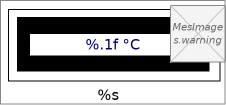
VISUALIZATION VISU_TEMPRO_PLUS_90  // 226x105
VAR_IN_OUT
	m_Input_RECHAUF : BLOCK_TEMPRO90_ANA;
END_VAR
    Rectangle (17,17 192x54), colour toggle: m_Input_RECHAUF.STATE_PowerOn
    Rectangle (8,9 212x72), invisible if: NOT (m_Input_RECHAUF.AUTOR_PowerOn_IHM OR m_Input_RECHAUF.AUTOR_PowerOff_IHM) OR NOT PRG_User.ACTU_USER.MAINTENANCE
        tap m_Input_RECHAUF.M_PowerOn
    Rectangle (88,85 41x20), "%s", text variable: m_Input_RECHAUF.MNEMO
    RoundedRectangle (29,33 168x23), "%.1f °C", text variable: m_Input_RECHAUF.STATE_Temp
    Image (170,5 56x57), invisible if: NOT m_Input_RECHAUF.STATE_Nok, image: MesImages.warning
END_VISUALIZATION

// ---- Visualizations/Symbole/STACKER/VISU_SUBSTRAT_NO_NUM.TcVIS
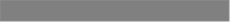
VISUALIZATION VISU_SUBSTRAT_NO_NUM  // 230x22
VAR_IN_OUT
	m_Input_MAP: STRUCT_MACHINE;
END_VAR
VAR_INPUT
	m_Input_NUM_CHAMBER : UDINT;
	m_Input_NUM_STATION : UDINT;
END_VAR
    Rectangle (0,0 228x20), invisible if: NOT m_Input_MAP.CHAMBER[m_Input_NUM_CHAMBER].STATION[m_Input_NUM_STATION].STATE_Unloaded
    Rectangle (0,0 228x20), invisible if: NOT m_Input_MAP.CHAMBER[m_Input_NUM_CHAMBER].STATION[m_Input_NUM_STATION].STATE_Loaded
    Rectangle (0,0 228x20), invisible if: m_Input_MAP.CHAMBER[m_Input_NUM_CHAMBER].STATION[m_Input_NUM_STATION].STATE_Loaded OR m_Input_MAP.CHAMBER[m_Input_NUM_CHAMBER].STATION[m_Input_NUM_STATION].STATE_Unloaded
END_VISUALIZATION

// ---- Visualizations/Symbole/VANNES/VISU_VANNE_2P_H.TcVIS
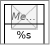
VISUALIZATION VISU_VANNE_2P_H  // 50x45
VAR_IN_OUT
	m_Input_VANNE : BLOCK_ACTUATOR;
END_VAR
    Rectangle (4,4 40x40), invisible if: TRUE
    Polygon (0,0)
    Rectangle (-1,25 50x20), "%s", text variable: m_Input_VANNE.MNEMO
    Polygon (0,0), colour toggle: (m_Input_VANNE.STATE_ON) <> 0, invisible if: NOT (m_Input_VANNE.STATE_OFF OR m_Input_VANNE.STATE_ON)
    Image (11,4 26x25), invisible if: NOT m_Input_VANNE.STATE_Nok, image: MesImages.warning
    Rectangle (4,4 40x20), invisible if: NOT (m_Input_VANNE.Autor_ON_IHM OR m_Input_VANNE.Autor_OFF_IHM) OR NOT PRG_User.ACTU_USER.MAINTENANCE
        tap m_Input_VANNE.M_ON
END_VISUALIZATION

// ---- Visualizations/Symbole/VANNES/VISU_VANNE_2P_H_ACT2.TcVIS
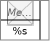
VISUALIZATION VISU_VANNE_2P_H_ACT2  // 50x41
VAR_IN_OUT
	m_Input_VANNE : BLOCK_ACTUATOR2;
END_VAR
    Rectangle (0,0 40x40), invisible if: TRUE
    Polygon (0,0)
    Rectangle (-5,21 50x20), "%s", text variable: m_Input_VANNE.MNEMO
    Polygon (0,0), colour toggle: (m_Input_VANNE.STATE_ON) <> 0, invisible if: NOT (m_Input_VANNE.STATE_OFF OR m_Input_VANNE.STATE_ON)
    Image (7,0 26x25), invisible if: NOT m_Input_VANNE.STATE_Nok, image: MesImages.warning
    Rectangle (0,0 40x20), invisible if: NOT (m_Input_VANNE.Autor_ON_IHM OR m_Input_VANNE.Autor_OFF_IHM) OR NOT PRG_User.ACTU_USER.MAINTENANCE
        tap m_Input_VANNE.M_ON
END_VISUALIZATION

// ---- Visualizations/Symbole/VANNES/VISU_VANNE_2P_V.TcVIS
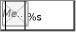
VISUALIZATION VISU_VANNE_2P_V  // 76x32
VAR_IN_OUT
	m_Input_VANNE : BLOCK_ACTUATOR;
END_VAR
    Rectangle (0,0 74x30), invisible if: TRUE
    Polygon (50,0)
    Polygon (50,0), colour toggle: (m_Input_VANNE.STATE_ON), invisible if: NOT (m_Input_VANNE.STATE_OFF OR m_Input_VANNE.STATE_ON) AND NOT PRG_USER.ACTU_USER.MAINTENANCE
    Rectangle (24,7 50x20), "%s", text variable: m_Input_VANNE.MNEMO
    Image (2,1 26x25), invisible if: NOT m_Input_VANNE.STATE_Nok, image: MesImages.warning
    Rectangle (5,0 20x30), invisible if: NOT (m_Input_VANNE.Autor_ON_IHM OR m_Input_VANNE.Autor_OFF_IHM) OR NOT PRG_User.ACTU_USER.MAINTENANCE
        tap m_Input_VANNE.M_ON
END_VISUALIZATION

// ---- Visualizations/Symbole/VANNES/VISU_VANNE_2P_V_ACT2.TcVIS
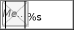
VISUALIZATION VISU_VANNE_2P_V_ACT2  // 74x30
VAR_IN_OUT
	m_Input_VANNE : BLOCK_ACTUATOR2;
END_VAR
    Rectangle (0,0 74x30), invisible if: TRUE
    Polygon (50,0)
    Polygon (50,0), colour toggle: (m_Input_VANNE.STATE_ON), invisible if: NOT (m_Input_VANNE.STATE_OFF OR m_Input_VANNE.STATE_ON) AND NOT PRG_USER.ACTU_USER.MAINTENANCE
    Rectangle (24,7 50x20), "%s", text variable: m_Input_VANNE.MNEMO
    Image (2,1 26x25), invisible if: NOT m_Input_VANNE.STATE_Nok, image: MesImages.warning
    Rectangle (5,0 20x30), invisible if: NOT (m_Input_VANNE.Autor_ON_IHM OR m_Input_VANNE.Autor_OFF_IHM) OR NOT PRG_User.ACTU_USER.MAINTENANCE
        tap m_Input_VANNE.M_ON
END_VISUALIZATION

// ---- Visualizations/Symbole/VANNES/VISU_VANNE_2P_V_NoPilot.TcVIS
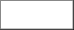
VISUALIZATION VISU_VANNE_2P_V_NoPilot  // 74x30
    Rectangle (0,0 74x30), invisible if: TRUE
    Polygon (50,0)
END_VISUALIZATION

// ---- Visualizations/Symbole/VANNES/VISU_VANNE_3P_H.TcVIS
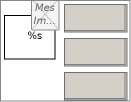
VISUALIZATION VISU_VANNE_3P_H  // 131x102
VAR_IN_OUT
	m_Input_Vanne	:	BLOCK_VVAT_3P;
END_VAR
    Rectangle (4,15 51x44), invisible if: TRUE
    Polygon (0,0), colour toggle: m_Input_Vanne.STATE_Lam
    Rectangle (13,25 44x21), "%s", text variable: m_Input_Vanne.MNEMO
    Polygon (0,0), colour toggle: m_Input_Vanne.STATE_On, invisible if: NOT (m_Input_Vanne.STATE_Off or m_Input_Vanne.STATE_On)
    Button (64,4 63x28), input disabled if: NOT m_Input_Vanne.AUTOR_On_IHM OR NOT .PRG_USER.ACTU_USER.MAINTENANCE, text list: 'TextList_VVAT_3P', text index: 0
        OnMouseClick: toggle m_Input_Vanne.M_On
    Button (64,38 63x28), input disabled if: NOT m_Input_Vanne.AUTOR_Lam_IHM OR NOT .PRG_USER.ACTU_USER.MAINTENANCE, text list: 'TextList_VVAT_3P', text index: 2
        OnMouseClick: toggle m_Input_Vanne.M_Lam
    Button (64,72 63x28), input disabled if: NOT m_Input_Vanne.AUTOR_Off_IHM OR NOT .PRG_USER.ACTU_USER.MAINTENANCE, text list: 'TextList_VVAT_3P', text index: 1
        OnMouseClick: toggle m_Input_Vanne.M_Off
    Image (31,-2 28x32), invisible if: NOT m_Input_Vanne.STATE_Nok, image: MesImages.warning
END_VISUALIZATION

// ---- Visualizations/Symbole/VANNES/VISU_VANNE_ASS_H.TcVIS
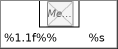
VISUALIZATION VISU_VANNE_ASS_H  // 118x49
VAR_IN_OUT
	m_Input_VANNE : BLOCK_VVAT_650_NO;
END_VAR

VAR_INPUT
	m_Input_NumFrame_Manu:	USINT;		(*numéro de frame à afficher dans le synoptique MANUEL*)
END_VAR
    Rectangle (0,0 118x49), invisible if: TRUE
    Polygon (0,0), colour toggle: m_Input_VANNE.STATE_Lam
    Rectangle (76,28 41x20), "%s", text variable: m_Input_VANNE.MNEMO
    Polygon (0,0), colour toggle: m_Input_VANNE.STATE_On, invisible if: NOT (m_Input_VANNE.STATE_Off OR m_Input_VANNE.STATE_On)
    Ellipse (54,2 10x10), colour toggle: m_Input_VANNE.STATE_Ok, invisible if: NOT m_Input_VANNE.STATE_Ok
    Rectangle (1,28 77x20), "%1.1f%%", text variable: m_Input_VANNE.STATE_Position
    Image (47,1 26x25), invisible if: NOT m_Input_VANNE.STATE_Nok, image: MesImages.warning
    Rectangle (39,0 40x27), invisible if: NOT m_Input_VANNE.MANUAL
        OnMouseClick: execute { .VISU_INDEX_MANU := m_Input_NumFrame_Manu; }
        OnMouseClick: change screen: SYN_MANUEL
END_VISUALIZATION

// ---- Visualizations/Symbole/VANNES/VISU_VANNE_ASS_H_MANU.TcVIS
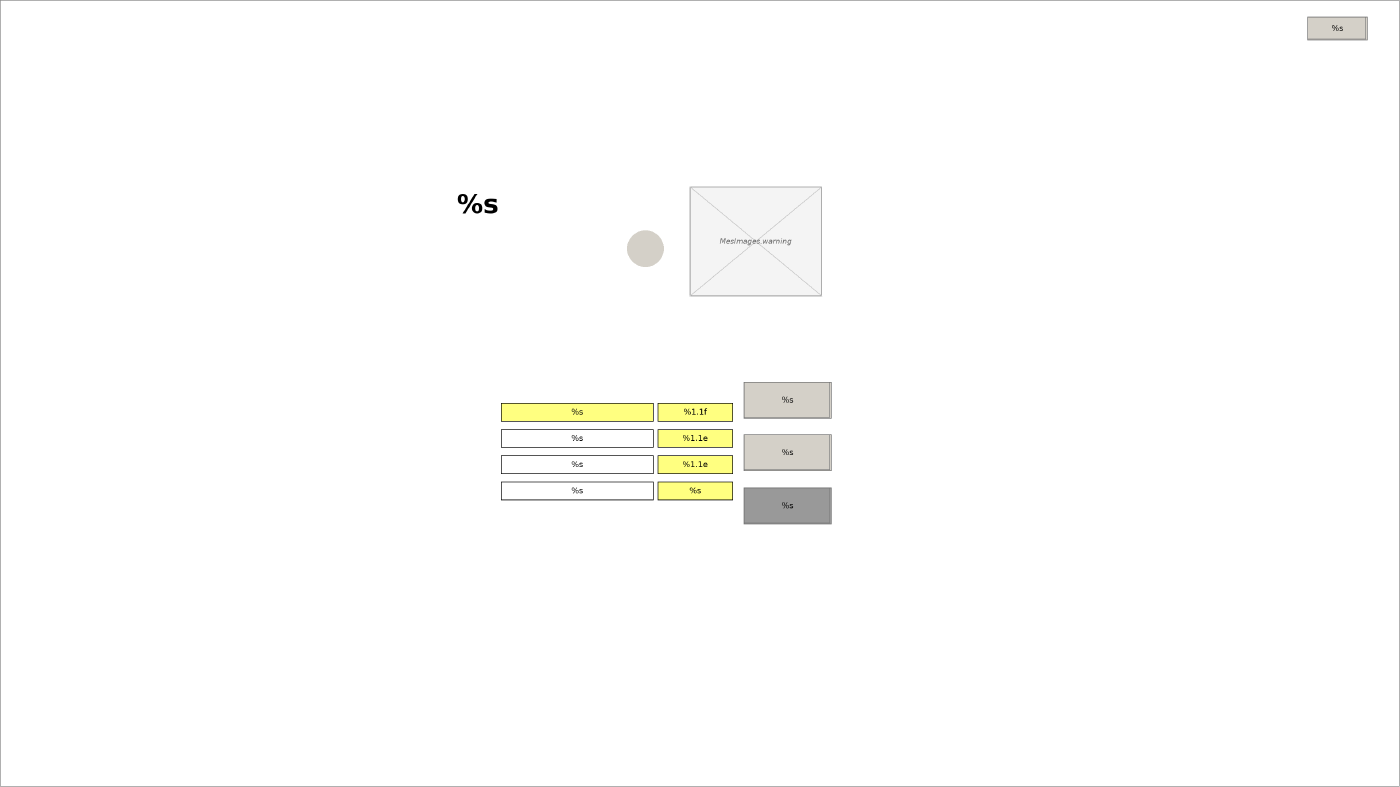
VISUALIZATION VISU_VANNE_ASS_H_MANU  // 1920x1080
VAR_IN_OUT
	m_Input_Vanne:		BLOCK_VVAT_650_NO;
	m_Input_State_Manu:	BOOL;
END_VAR
    Button (1793,23 82x32), "%s", text list: 'TextList_Basiques', text index: 8
        OnMouseClick: change screen: Previous 
        OnMouseClick: execute { .VISU_INDEX_MANU := 0; }
    Polygon (0,0), colour toggle: m_Input_VANNE.STATE_Lam
    Rectangle (573,246 165x68), "%s", text variable: m_Input_VANNE.MNEMO
    Polygon (0,0), colour toggle: m_Input_VANNE.STATE_On, invisible if: NOT (m_Input_VANNE.STATE_Off OR m_Input_VANNE.STATE_On)
    Ellipse (860,316 50x50), colour toggle: m_Input_VANNE.STATE_Ok
    Image (946,256 181x150), invisible if: NOT m_Input_VANNE.STATE_Nok, image: MesImages.warning
    Button (1020,524 120x50), "%s", input disabled if: NOT m_Input_Vanne.AUTOR_On_IHM OR NOT .PRG_USER.ACTU_USER.MAINTENANCE, text list: 'TextList_VVAT_3P', text index: 0
        toggle m_Input_Vanne.M_On
    Button (1020,596 120x50), "%s", input disabled if: NOT m_Input_Vanne.AUTOR_Off_IHM OR NOT .PRG_USER.ACTU_USER.MAINTENANCE, text list: 'TextList_VVAT_3P', text index: 1
        toggle m_Input_Vanne.M_Off
    Button (1020,669 120x50), "%s", input disabled if: NOT m_Input_Vanne.AUTOR_Lam_IHM OR NOT .PRG_USER.ACTU_USER.MAINTENANCE, text list: 'TextList_VVAT_3P', text index: 2
        toggle m_Input_Vanne.M_Lam
    RoundedRectangle (687,553 209x25), "%s", invisible if: NOT m_Input_Vanne.PRM_Mode, input disabled if: NOT .PRG_USER.ACTU_USER.MAINTENANCE OR NOT m_Input_State_Manu OR NOT m_Input_Vanne.PRM_Mode, text list: 'TextList_VVAT_650_ETHERCAT', text index: 8
        OnMouseClick: toggle m_Input_Vanne.PRM_Mode
    RoundedRectangle (687,553 209x25), "%s", invisible if: m_Input_Vanne.PRM_Mode, input disabled if: NOT .PRG_USER.ACTU_USER.MAINTENANCE OR NOT m_Input_State_Manu OR m_Input_Vanne.PRM_Mode, text list: 'TextList_VVAT_650_ETHERCAT', text index: 7
        OnMouseClick: toggle m_Input_Vanne.PRM_Mode
    RoundedRectangle (687,589 209x25), "%s", invisible if: NOT m_Input_Vanne.PRM_Mode, text list: 'TextList_VVAT_650_ETHERCAT', text index: 4
    RoundedRectangle (687,625 209x25), "%s", invisible if: NOT m_Input_Vanne.PRM_Mode, text list: 'TextList_VVAT_650_ETHERCAT', text index: 5
    RoundedRectangle (687,661 209x25), "%s", invisible if: NOT m_Input_Vanne.PRM_Mode, text list: 'TextList_VVAT_650_ETHERCAT', text index: 6
    RoundedRectangle (902,661 103x25), "%s", text variable: m_Input_Vanne.PRM_Tim_W_Pr, invisible if: NOT m_Input_Vanne.PRM_Mode, input disabled if: NOT m_Input_Vanne.PRM_Mode
        OnMouseClick: write the text variable via Edit
    RoundedRectangle (902,625 103x25), "%1.1e", text variable: m_Input_Vanne.PRM_W_Pr_HI, invisible if: NOT m_Input_Vanne.PRM_Mode, input disabled if: NOT m_Input_Vanne.PRM_Mode
        OnMouseClick: write the text variable via InputWithLimits, min 0, max 1000
    RoundedRectangle (902,589 103x25), "%1.1e", text variable: m_Input_Vanne.PRM_W_Pr_LO, invisible if: NOT m_Input_Vanne.PRM_Mode, input disabled if: NOT m_Input_Vanne.PRM_Mode
        OnMouseClick: write the text variable via InputWithLimits, min 0, max 1000
    RoundedRectangle (902,553 103x25), "%1.1e", text variable: m_Input_Vanne.PRM_Pression, invisible if: NOT m_Input_Vanne.PRM_Mode, input disabled if: NOT m_Input_Vanne.PRM_Mode
        OnMouseClick: write the text variable via InputWithLimits, min 0, max 1000
    RoundedRectangle (902,553 103x25), "%1.1f", text variable: m_Input_Vanne.PRM_Position, invisible if: m_Input_Vanne.PRM_Mode, input disabled if: m_Input_Vanne.PRM_Mode
        OnMouseClick: write the text variable via InputWithLimits, min 0, max 100
END_VISUALIZATION

// ---- Visualizations/Symbole/VANNES/VISU_VANNE_ASS_VAT653_ETHERCAT.TcVIS
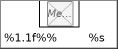
VISUALIZATION VISU_VANNE_ASS_VAT653_ETHERCAT  // 118x49
VAR_IN_OUT
	m_Input_VANNE : BLOCK_VVAT_653_ETHERCAT;
END_VAR

VAR_INPUT
	m_Input_NumFrame_Manu:	USINT;		(*numéro de frame à afficher dans le synoptique MANUEL*)
END_VAR
    Rectangle (0,0 118x49), invisible if: TRUE
    Polygon (0,0), colour toggle: m_Input_VANNE.STATE_Lam
    Rectangle (76,28 41x20), "%s", text variable: m_Input_VANNE.MNEMO
    Polygon (0,0), colour toggle: m_Input_VANNE.STATE_On, invisible if: NOT (m_Input_VANNE.STATE_Off OR m_Input_VANNE.STATE_On)
    Ellipse (54,2 10x10), colour toggle: m_Input_VANNE.STATE_Ok, invisible if: NOT m_Input_VANNE.STATE_Ok
    Rectangle (1,28 77x20), "%1.1f%%", text variable: m_Input_VANNE.STATE_Position
    Image (47,1 26x25), invisible if: NOT m_Input_VANNE.STATE_Nok, image: MesImages.warning
    Rectangle (39,0 40x27), invisible if: NOT m_Input_VANNE.MANUAL
        OnMouseClick: execute { .VISU_INDEX_MANU := m_Input_NumFrame_Manu; }
        OnMouseClick: change screen: SYN_MANUEL
END_VISUALIZATION

// ---- Visualizations/Symbole/VANNES/VISU_VANNE_ASS_VAT653_ETHERCAT_MANU.TcVIS
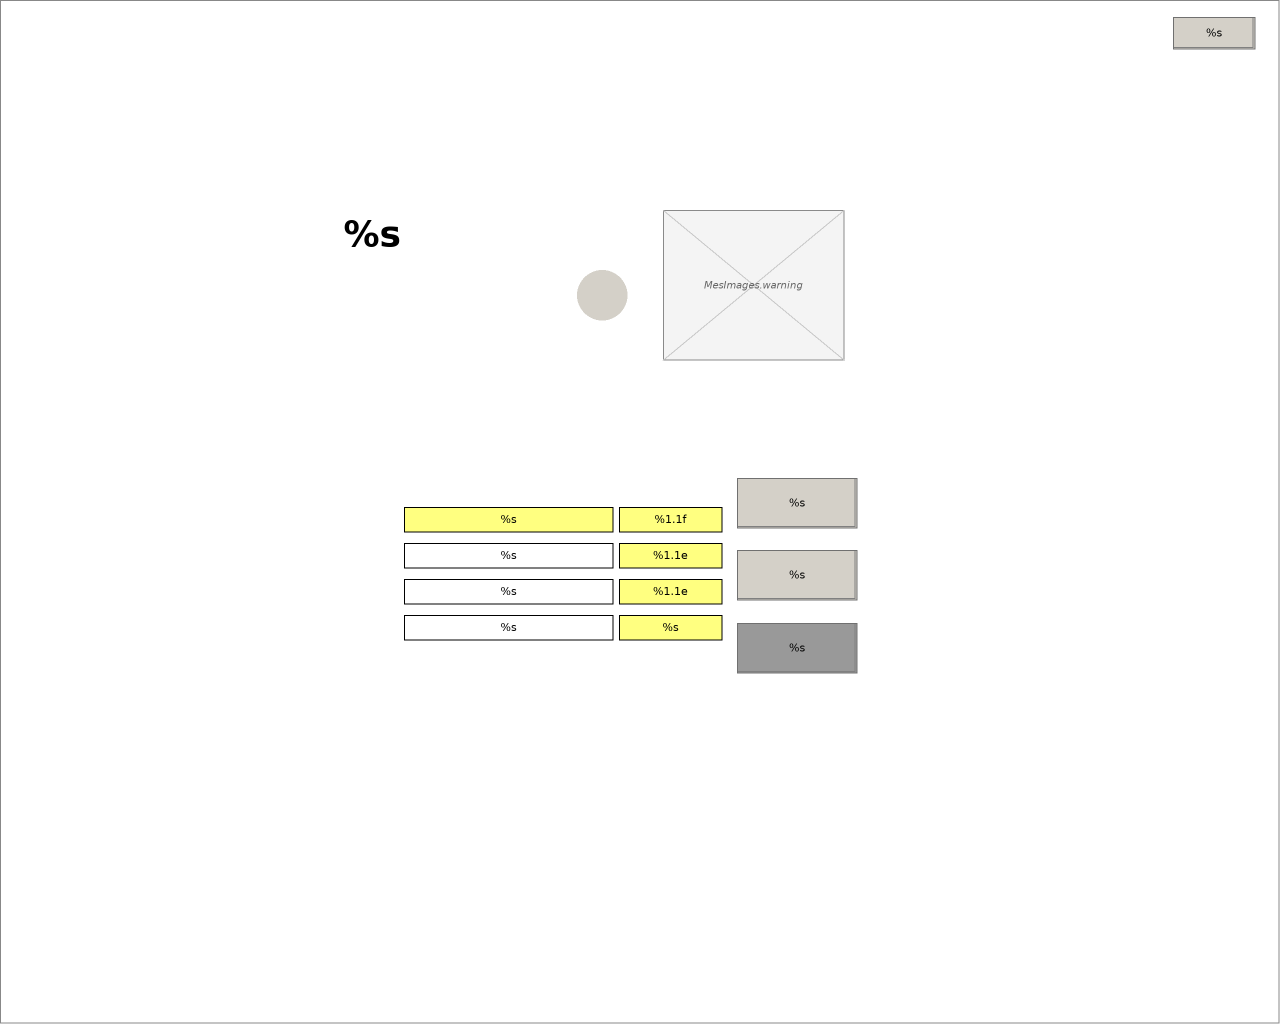
VISUALIZATION VISU_VANNE_ASS_VAT653_ETHERCAT_MANU  // 1280x1024
VAR_IN_OUT
	m_Input_Vanne:		BLOCK_VVAT_653_ETHERCAT;
	m_Input_State_Manu:	BOOL;
END_VAR
    Button (1173,17 82x32), "%s", text list: 'TextList_Basiques', text index: 8
        OnMouseClick: change screen: Previous 
        OnMouseClick: execute { .VISU_INDEX_MANU := 0; }
    Polygon (0,0), colour toggle: m_Input_VANNE.STATE_Lam
    Rectangle (290,200 165x68), "%s", text variable: m_Input_VANNE.MNEMO
    Polygon (0,0), colour toggle: m_Input_VANNE.STATE_On, invisible if: NOT (m_Input_VANNE.STATE_Off OR m_Input_VANNE.STATE_On)
    Ellipse (577,270 50x50), colour toggle: m_Input_VANNE.STATE_Ok, invisible if: NOT m_Input_VANNE.STATE_Ok
    Image (663,210 181x150), invisible if: NOT m_Input_VANNE.STATE_Nok, image: MesImages.warning
    Button (737,478 120x50), "%s", input disabled if: NOT m_Input_Vanne.AUTOR_On_IHM OR NOT .PRG_USER.ACTU_USER.MAINTENANCE, text list: 'TextList_VVAT_3P', text index: 0
        toggle m_Input_Vanne.M_On
    Button (737,550 120x50), "%s", input disabled if: NOT m_Input_Vanne.AUTOR_Off_IHM OR NOT .PRG_USER.ACTU_USER.MAINTENANCE, text list: 'TextList_VVAT_3P', text index: 1
        toggle m_Input_Vanne.M_Off
    Button (737,623 120x50), "%s", input disabled if: NOT m_Input_Vanne.AUTOR_Lam_IHM OR NOT .PRG_USER.ACTU_USER.MAINTENANCE, text list: 'TextList_VVAT_3P', text index: 2
        toggle m_Input_Vanne.M_Lam
    RoundedRectangle (404,507 209x25), "%s", invisible if: NOT m_Input_Vanne.PRM_Mode, input disabled if: NOT .PRG_USER.ACTU_USER.MAINTENANCE OR NOT m_Input_State_Manu OR NOT m_Input_Vanne.PRM_Mode, text list: 'TextList_VVAT_650_ETHERCAT', text index: 8
        OnMouseClick: toggle m_Input_Vanne.PRM_Mode
    RoundedRectangle (404,507 209x25), "%s", invisible if: m_Input_Vanne.PRM_Mode, input disabled if: NOT .PRG_USER.ACTU_USER.MAINTENANCE OR NOT m_Input_State_Manu OR m_Input_Vanne.PRM_Mode, text list: 'TextList_VVAT_650_ETHERCAT', text index: 7
        OnMouseClick: toggle m_Input_Vanne.PRM_Mode
    RoundedRectangle (404,543 209x25), "%s", invisible if: NOT m_Input_Vanne.PRM_Mode, text list: 'TextList_VVAT_650_ETHERCAT', text index: 4
    RoundedRectangle (404,579 209x25), "%s", invisible if: NOT m_Input_Vanne.PRM_Mode, text list: 'TextList_VVAT_650_ETHERCAT', text index: 5
    RoundedRectangle (404,615 209x25), "%s", invisible if: NOT m_Input_Vanne.PRM_Mode, text list: 'TextList_VVAT_650_ETHERCAT', text index: 6
    RoundedRectangle (619,615 103x25), "%s", text variable: m_Input_Vanne.PRM_Tim_W_Pr, invisible if: NOT m_Input_Vanne.PRM_Mode, input disabled if: NOT m_Input_Vanne.PRM_Mode
        OnMouseClick: write the text variable via VisuDialogs.Keypad
    RoundedRectangle (619,579 103x25), "%1.1e", text variable: m_Input_Vanne.PRM_W_Pr_HI, invisible if: NOT m_Input_Vanne.PRM_Mode, input disabled if: NOT m_Input_Vanne.PRM_Mode
        OnMouseClick: write the text variable via VisuDialogs.NumpadExtended, min 0, max 1000
    RoundedRectangle (619,543 103x25), "%1.1e", text variable: m_Input_Vanne.PRM_W_Pr_LO, invisible if: NOT m_Input_Vanne.PRM_Mode, input disabled if: NOT m_Input_Vanne.PRM_Mode
        OnMouseClick: write the text variable via VisuDialogs.NumpadExtended, min 0, max 1000
    RoundedRectangle (619,507 103x25), "%1.1e", text variable: m_Input_Vanne.PRM_Pression, invisible if: NOT m_Input_Vanne.PRM_Mode, input disabled if: NOT m_Input_Vanne.PRM_Mode
        OnMouseClick: write the text variable via VisuDialogs.NumpadExtended, min 0, max 1000
    RoundedRectangle (619,507 103x25), "%1.1f", text variable: m_Input_Vanne.PRM_Position, invisible if: m_Input_Vanne.PRM_Mode, input disabled if: m_Input_Vanne.PRM_Mode
        OnMouseClick: write the text variable via VisuDialogs.Numpad, min 0, max 100
END_VISUALIZATION

// ---- Visualizations/Synoptique/SYN_EXEC_PROC.TcVIS
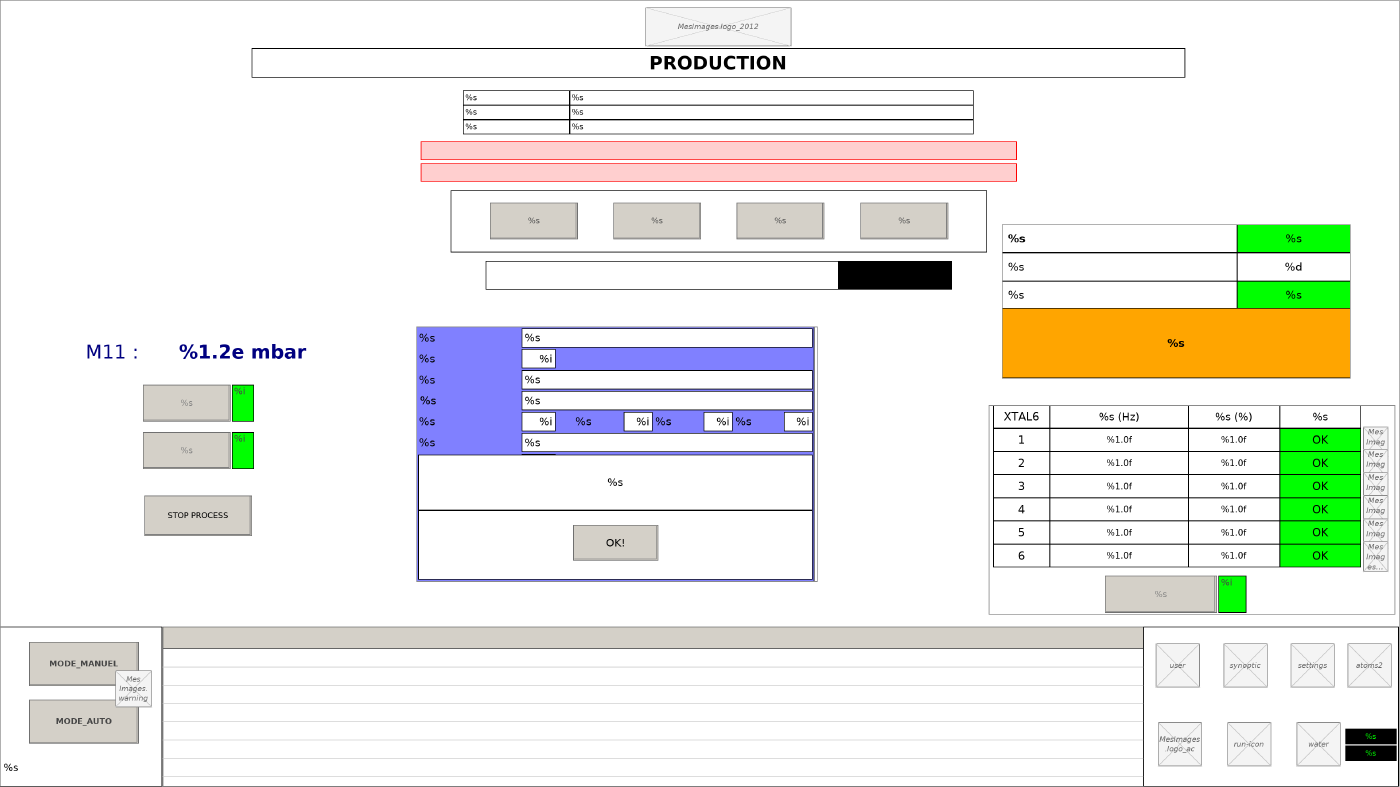
VISUALIZATION SYN_EXEC_PROC  // 1920x1080, background image fond_blanc_1280_1024
    Frame (223,860 1346x161)
        shows VISU_EV_EXTRAIT()
    Frame (1568,860 352x162)
        shows VISU_BANDEAU(m_Input_MACHINE := Global_Variables.MACHINE)
    Frame (0,860 221x162)
        shows VISU_MODE_MARCHE(m_Input_MACHINE := .MACHINE)
    RoundedRectangle (345,66 1280x40), "PRODUCTION"
    Group (635,124 700x60)
        Rectangle (0,0 146x20), "%s", text list: 'TextList_Process', text index: 0
        Rectangle (0,20 146x20), "%s", text list: 'TextList_Process', text index: 1
        Rectangle (0,40 146x20), "%s", text list: 'TextList_Process', text index: 2
        Rectangle (146,0 554x20), "%s", text variable: EXECPROC.PRM_PROCESS_NAME, text index: 0
        Rectangle (146,20 554x20), "%s", text variable: EXECPROC.STATE_STEP_TEXT, text index: 0
        Rectangle (146,40 554x20), "%s", text variable: MAIN.STEP_EMPILEMENT.STATE_LAYER_TEXT, text index: 0
    Group (618,261 735x85)
        RoundedRectangle (0,0 735x85)
        Button (54,17 120x50), "%s", input disabled if: (NOT MACHINE.AUTOR_Start_Prod_Ihm OR PRG_SEC.VERROU OR NOT PRG_User.ACTU_USER.PRODUCTION) OR MACHINE.STATE_Prod, text list: 'TextList_Process', text index: 3
            tap MAIN.bStartVerif
        Button (223,17 120x50), "%s", input disabled if: NOT (PRG_USER.ACTU_USER.PRODUCTION AND MACHINE.AUTOR_Stop_Prod_Ihm), text list: 'TextList_Process', text index: 4
            toggle MACHINE.M_Stop_Prod
        Button (392,17 120x50), "%s", input disabled if: NOT (PRG_USER.ACTU_USER.PRODUCTION AND MACHINE.AUTOR_Inter_Prod_ihm), text list: 'TextList_Process', text index: 5
            toggle MACHINE.M_inter_Prod
        Button (562,17 120x50), "%s", input disabled if: NOT (PRG_USER.ACTU_USER.PRODUCTION AND MACHINE.AUTOR_Repris_Prod_ihm), text list: 'TextList_Process', text index: 6
            toggle MACHINE.M_Reprise_Prod
    Frame (571,448 550x350), invisible if: NOT Global_Variables.MACHINE.STATE_Prod
        shows VISU_INFO_PROCESS()
    Image (885,10 200x53), image: MesImages.logo_2012
    Frame (196,528 153x52)
        shows VISU_FCTS_SA(m_Input_ID_XML := 4, m_Input_UserRight := PRG_USER.ACTU_USER.PRODUCTION AND NOT MACHINE.STATE_Prod AND NOT INIT_MACHINE.OP_INIT.EC, m_Input_Operation := PRG_POMPAGE.POMPAGE.OP_Ventilation)
    Frame (196,593 153x52)
        shows VISU_FCTS_SA(m_Input_ID_XML := 0, m_Input_UserRight := PRG_USER.ACTU_USER.PRODUCTION AND NOT MACHINE.STATE_Prod AND NOT INIT_MACHINE.OP_INIT.EC, m_Input_Operation := PRG_POMPAGE.POMPAGE.OP_Pompage_Sec)
    Button (198,680 147x55), "STOP PROCESS", invisible if: PRG_USER.ACTU_USER.MAINTENANCE OR NOT INIT_MACHINE.STATE_ABORT
        tap INIT_MACHINE.M_Stop_Procedure
    Group (666,358 639x39)
        Rectangle (0,0 484x39), text list: 'TextList_EcoMode', text index: 12
        Rectangle (484,0 155x39), colour toggle: MACHINE.PRM_EXEC_PROC_WEEKEND, input disabled if: NOT Global_Variables.PRG_USER.ACTU_USER.PRODUCTION
            toggle MACHINE.PRM_EXEC_PROC_WEEKEND
    Frame (1374,308 478x211)
        shows VISU_MODE_QUARTZ(m_input_Mode_Quartz := MODE_QUARTZ_PROD)
    Frame (1356,556 557x287)
        shows VISU_XTAL6_PROD(m_Input_XTAL6 := PRG_EVAP.QZ1)
    Rectangle (114,463 80x40), "M11 :"
    Rectangle (208,463 250x40), "%1.2e mbar", text variable: Global_Variables.PRG_POMPAGE.M11.STATE_Pression
    Group (577,194 817x55)
        Rectangle (0,0 817x25), invisible if: NOT MACHINE.DEF_Presence_TrAC.DEF, text list: 'TextList_Basiques', text index: 20
        Rectangle (0,30 817x25), invisible if: NOT MACHINE.DEF_Presence_ACSoft.DEF, text list: 'TextList_Basiques', text index: 21
END_VISUALIZATION

// ---- Visualizations/Synoptique/SYN_INFOS.TcVIS
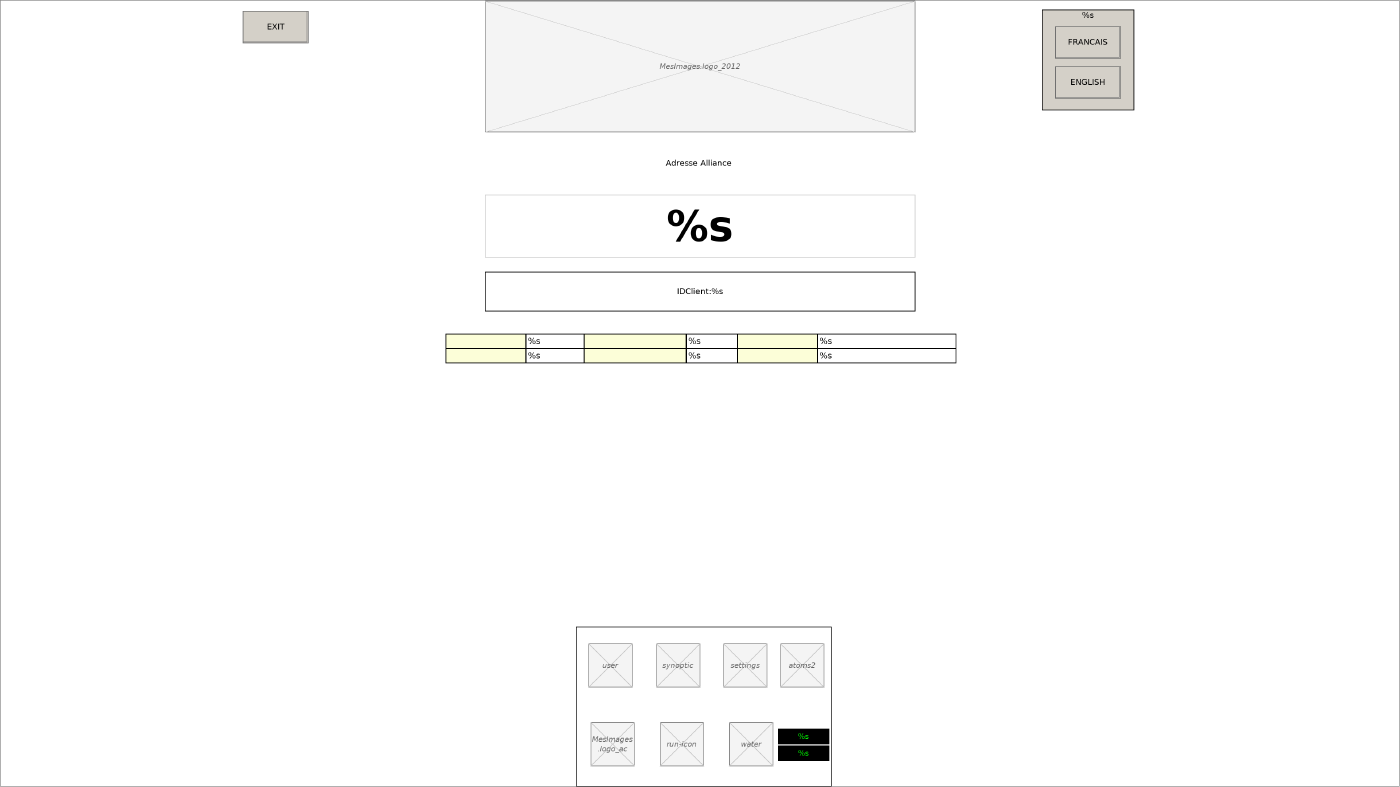
VISUALIZATION SYN_INFOS  // 1920x1080
    Image (665,1 590x180), image: MesImages.logo_2012
    Textfield (665,181 590x86), "Adresse Alliance"
    Textfield (665,267 590x86), "%s", text variable: MACHINE.CONF_Name
    RoundedRectangle (665,373 590x54), "IDClient:%s", text variable: MACHINE.CONF_Customer
    Rectangle (611,458 110x20), text list: 'TextList_Infos', text index: 1
    Rectangle (721,458 80x20), "%s", text variable: Global_Variables.MACHINE.CONF_Affaire
    Rectangle (611,478 110x20), text list: 'TextList_Infos', text index: 2
    Rectangle (721,478 80x20), "%s", text variable: Global_Variables.MACHINE.CONF_Author
    Rectangle (801,478 140x20), text list: 'TextList_Infos', text index: 4
    Rectangle (941,458 70x20), "%s", text variable: Global_Variables.MACHINE.CONF_Version
    Rectangle (801,458 140x20), text list: 'TextList_Infos', text index: 3
    Rectangle (941,478 70x20), "%s", text variable: Global_Variables.MACHINE.CONF_VerDate
    Rectangle (1011,478 110x20), text list: 'TextList_Infos', text index: 6
    Rectangle (1121,458 190x20), "%s", text variable: Global_Variables.MACHINE.CONF_SerialNumber
    Rectangle (1011,458 110x20), text list: 'TextList_Infos', text index: 5
    Rectangle (1121,478 190x20), "%s", text variable: Global_Variables.MACHINE.CONF_Model
    RoundedRectangle (1429,13 126x138), "%s", text list: 'TextList_Infos', text index: 0
    Button (1447,36 90x44), "FRANCAIS"
        OnMouseClick: ChangeLanguage ChangeLanguage=FR
    Button (1447,91 90x44), "ENGLISH"
        OnMouseClick: ChangeLanguage ChangeLanguage=EN
    Frame (790,860 352x220)
        shows VISU_BANDEAU(m_Input_MACHINE := Global_Variables.MACHINE)
    Button (333,15 90x44), "EXIT", text list: ''
        OnMouseClick: change screen: SYN_PROC
        OnMouseDown: ExecuteCommand ExecuteCommand=ExecuteCommand=[Command=ExecuteClientProgram, Value='C:\Machine\PLC\Exit_TC3Hmi.bat']
END_VISUALIZATION

// ---- Visualizations/Synoptique/SYN_MANUEL.TcVIS
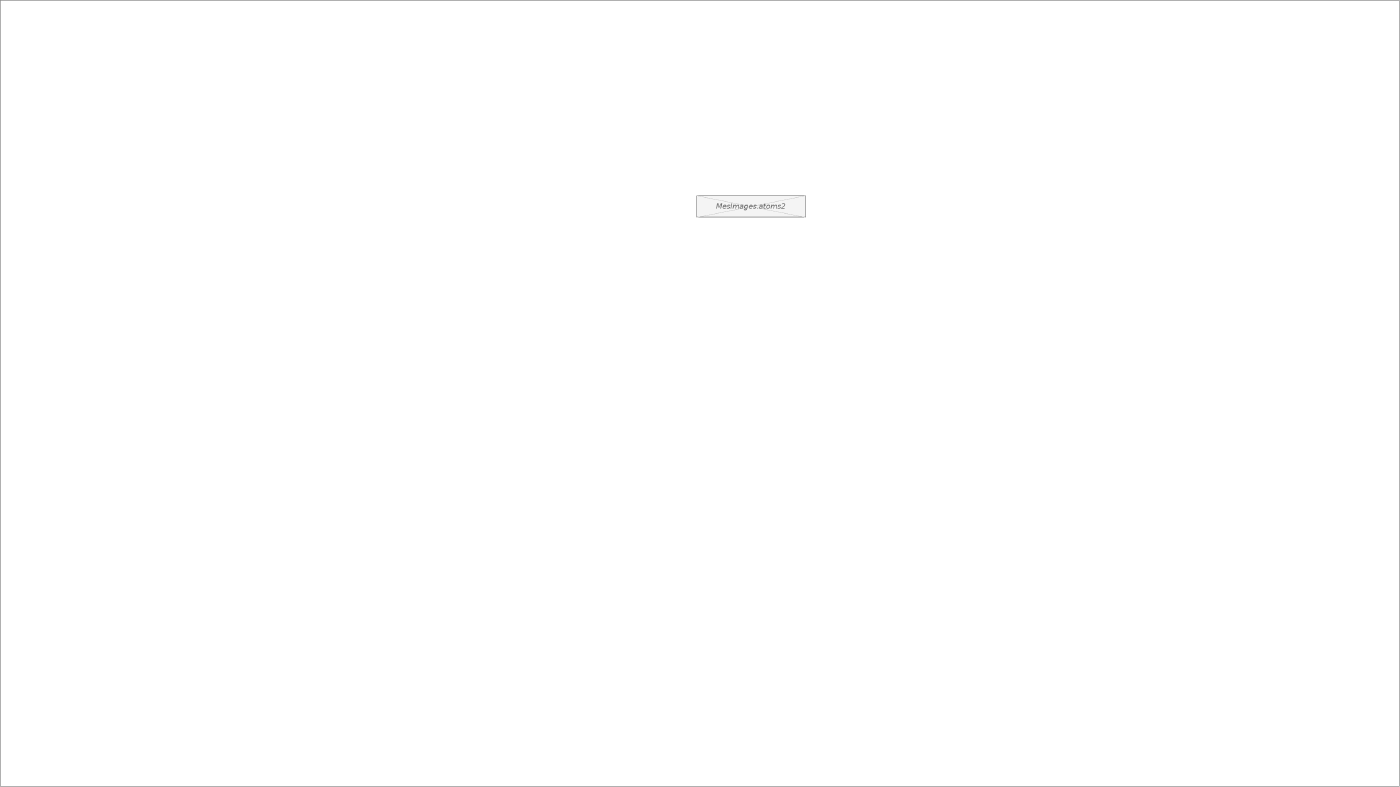
VISUALIZATION SYN_MANUEL  // 1920x1080, background image fond_blanc_1280_1024
    Frame (0,0 1920x1080), frame switch variable: VISU_INDEX_MANU
        shows VISU_BLANCK_MANUEL()
        shows VISU_XTAL6_ZOOM(m_Input_XTAL6 := .PRG_EVAP.QZ1)
        shows VISU_INFO(m_Input_CRYO := PRG_POMPAGE.COM_CRYOS, m_Input_PRG_POMPAGE := PRG_POMPAGE)
        shows VISU_VANNE_ASS_H_MANU(m_Input_Vanne := PRG_POMPAGE.POMPAGE.VS11, m_Input_State_Manu := MACHINE.STATE_Manu)
        [2]: m_Input_ID_NOM_XML=10, m_Input_INDEX_MOTEUR=2, m_Input_Ref_Trf=0
        p2655817705: .PRG_PUISSANCE.RF1
        p3040719188: .ENCEINTE.STATE_Manu
        p4051230613: PRG_MOUVEMENT_PS.ROTATION_PS
        p3521815518: PRG_MOUVEMENT_PS.TILT_PS
        p625233746: PRG_MOUVEMENT_PS.ROTATION_PS
    Image (955,268 150x30), image: MesImages.atoms2
END_VISUALIZATION

// ---- Visualizations/Synoptique/SYN_POMPAGE.TcVIS
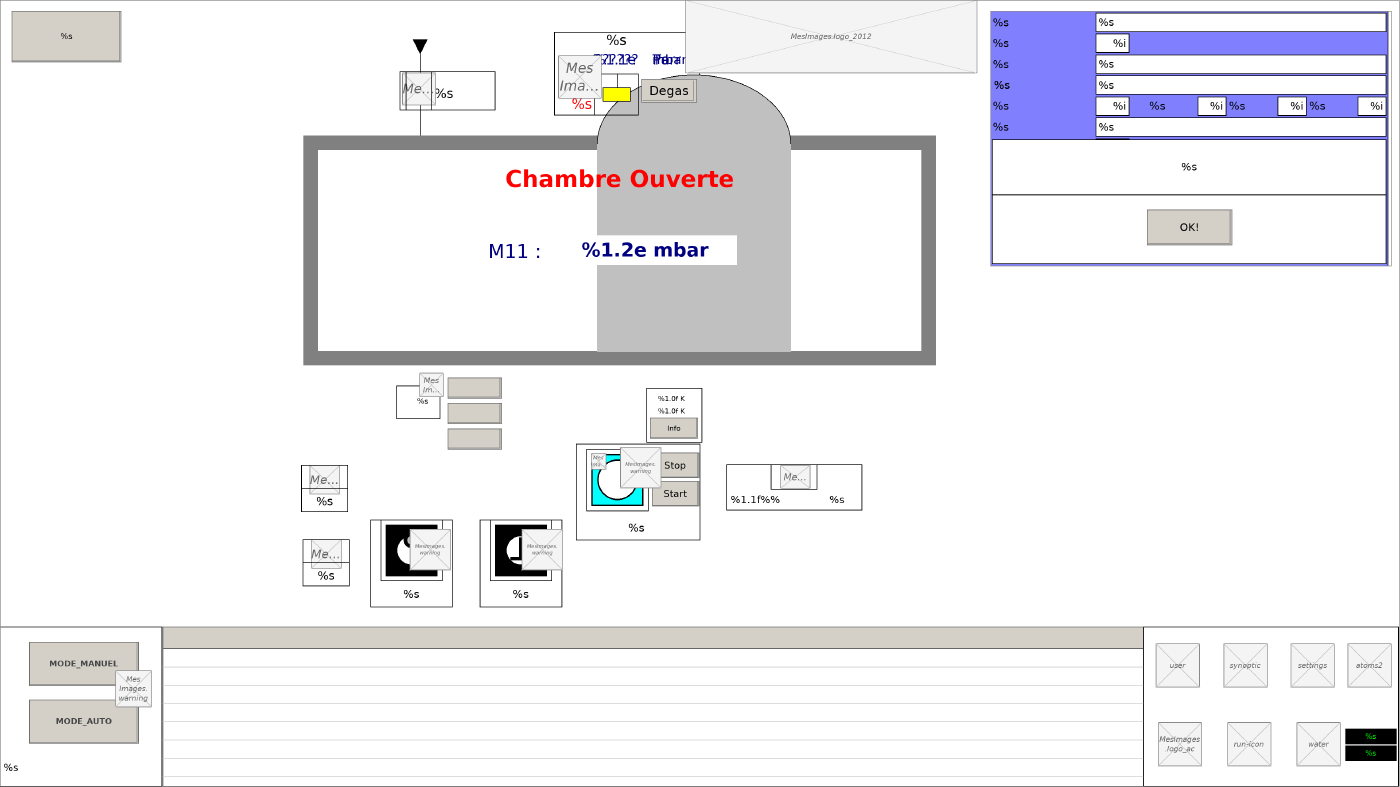
VISUALIZATION SYN_POMPAGE  // 1920x1080, background image fond_blanc_1280_1024
    Frame (223,860 710x161)
        shows VISU_EV_EXTRAIT()
    Frame (1568,860 352x162)
        shows VISU_BANDEAU(m_Input_MACHINE := Global_Variables.MACHINE)
    Frame (0,860 221x162)
        shows VISU_MODE_MARCHE(m_Input_MACHINE := .MACHINE)
    Button (16,15 150x70), "%s", text list: 'TextList_Navigation', text index: 1
        OnMouseClick: change screen: SYN_PROC
    Line (846,102) (846,217)
    Line (576,62) (576,216)
    RoundedRectangle (416,186 867x315)
    Frame (760,44 200x114)
        shows VISU_JAUGE_BCG450_V_HAUT_ETHERCAT(m_Input_JAUGE := PRG_POMPAGE.M11)
    Frame (548,98 135x60)
        shows VISU_VANNE_2P_V(m_Input_VANNE := PRG_POMPAGE.POMPAGE.VH11)
    Polygon (566,54) (586,54) (576,74)
    Rectangle (666,325 80x40), "M11 :"
    Rectangle (760,323 250x40), "%1.2e mbar", text variable: Global_Variables.PRG_POMPAGE.M11.STATE_Pression
    Label (669,214 362x63), "Chambre Ouverte", invisible if: PRG_POMPAGE.IN_FE11T
    Frame (1358,15 550x350), invisible if: NOT Global_Variables.MACHINE.STATE_Prod
        shows VISU_INFO_PROCESS()
    Polyline (458,705)
    Polyline (330,705)
    Polygon (337,745)
    Frame (407,632 80x80)
        shows VISU_VANNE_2P_H(m_Input_VANNE := PRG_POMPAGE.POMPAGE.VINT)
    Polyline (840,705)
    Frame (790,609 170x177)
        shows VISU_POMPE_CRYO_CTI(m_Input_POMPE := PRG_POMPAGE.POMPAGE.PS11, m_Input_COM := PRG_POMPAGE.COM_CRYOS, m_Input_Forcage := PRG_POMPAGE.POMPAGE.PS11.PRM_Forcage_Cryo_EXT)
    Polyline (553,751)
    Frame (884,532 100x75)
        shows VISU_TEMP_POMP_CRYO_SOLO(m_Input_CRYO := PRG_POMPAGE.COM_CRYOS, m_Input_PRG_POMPAGE := PRG_POMPAGE, m_Input_NumFrame_Manu := 2, m_Input_INDEX_CRYO := 1)
    Rectangle (170,643 200x30), text list: 'TextList_Pompage', text index: 0
    Polyline (458,664)
    Frame (508,713 120x120)
        shows VISU_POMPE_PRIMAIRE(m_Input_POMPE := PRG_POMPAGE.POMPAGE.PP11)
    Frame (658,713 120x120)
        shows VISU_POMPE_ROOTS(m_Input_POMPE := PRG_POMPAGE.POMPAGE.PR11)
    Frame (409,734 80x80)
        shows VISU_VANNE_2P_H(m_Input_VANNE := PRG_POMPAGE.POMPAGE.VN2PP11)
    Polygon (337,745)
    Image (940,0 400x100), image: MesImages.logo_2012
    Frame (539,514 154x105)
        shows VISU_VANNE_3P_H(m_Input_Vanne := PRG_POMPAGE.POMPAGE.VP11)
    Frame (996,637 186x63)
        shows VISU_VANNE_ASS_H(m_Input_VANNE := PRG_POMPAGE.POMPAGE.VS11, m_Input_NumFrame_Manu := 3)
END_VISUALIZATION

// ---- Visualizations/Synoptique/SYN_PROC.TcVIS
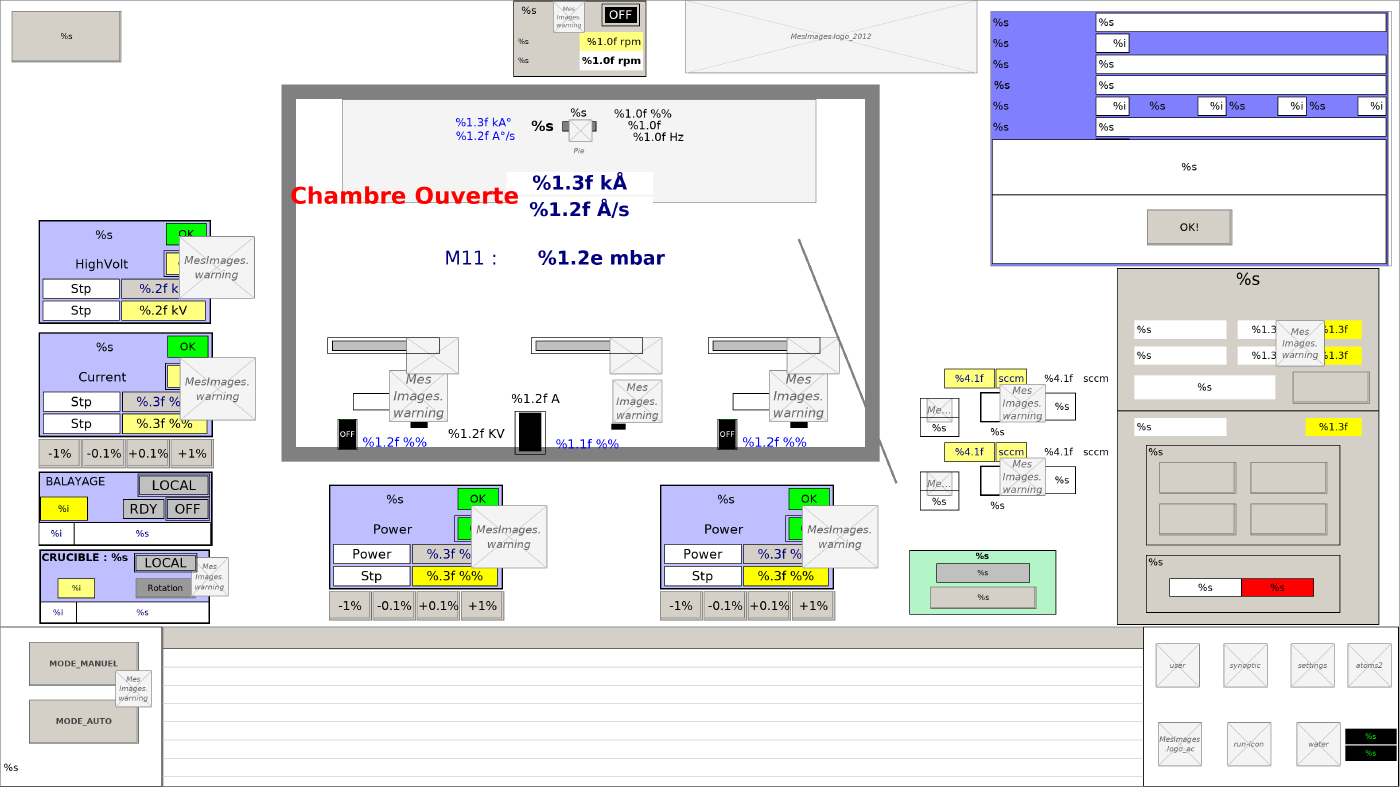
VISUALIZATION SYN_PROC  // 1920x1080, background image fond_blanc_1280_1024
    Frame (1239,746 216x103)
        shows VISU_ECOMODE()
    RoundedRectangle (386,116 820x517)
    Frame (704,1 182x104)
        shows VISU_ROT(m_Input_ROT := PRG_MOUVEMENT_PS.ROTATION_PS)
    Pie (469,136 650x142)
    Frame (223,860 710x161)
        shows VISU_EV_EXTRAIT()
    Frame (1568,860 352x162)
        shows VISU_BANDEAU(m_Input_MACHINE := Global_Variables.MACHINE)
    Rectangle (695,236 200x30), "%1.3f kÅ", text variable: PRG_EVAP.XTC3.STATE_Thickness
    Rectangle (695,270 200x35), "%1.2f Å/s", text variable: PRG_EVAP.XTC3.STATE_Rate
    Frame (0,860 221x162)
        shows VISU_MODE_MARCHE(m_Input_MACHINE := .MACHINE)
    Frame (603,140 400x84)
        shows VISU_XTAL_6(m_Input_XTAL := PRG_EVAP.QZ1, m_Input_NumFrame_Manu := 1)
    Button (16,15 150x70), "%s", text list: 'TextList_Navigation', text index: 0
        OnMouseClick: change screen: SYN_POMPAGE
    Frame (1532,368 360x489)
        shows VISU_XTC(M_Input_Evap := .PRG_EVAP.EVAPS1, M_Input_Ctrl := .PRG_EVAP.XTC3, M_Input_QZ1 := .PRG_EVAP.QZ1)
    Frame (1358,15 550x350), invisible if: NOT Global_Variables.MACHINE.STATE_Prod
        shows VISU_INFO_PROCESS()
    Frame (458,496 160x130)
        shows VISU_SOURCE_EFFET_JOULE(m_Input_SOURCE := PRG_EVAP.SOURCE2)
    Frame (451,665 300x186)
        shows VISU_CANON(m_Input_SOURCE := PRG_EVAP.SOURCE2)
    Frame (979,496 160x130)
        shows VISU_SOURCE_EFFET_JOULE(m_Input_SOURCE := PRG_EVAP.SOURCE3)
    Frame (905,665 300x186)
        shows VISU_CANON(m_Input_SOURCE := PRG_EVAP.SOURCE3)
    Frame (53,456 300x186)
        shows VISU_CANON_ST10(m_Input_SOURCE := .PRG_EVAP.SOURCE1)
    Frame (53,302 296x150)
        shows VISU_HT_CANON_ST10(m_Input_SOURCE := PRG_EVAP.SOURCE1)
    Frame (681,511 227x115)
        shows VISU_SOURCE_EVAP_COTE_ST10(m_Input_NO_IFIL_RET := FALSE, m_Input_NO_IEMISS_RET := FALSE, m_Input_SOURCE := PRG_EVAP.SOURCE1)
    Frame (728,463 180x50)
        shows SYM_CACHE(m_Input_CACHE := PRG_EVAP.CC11)
    Frame (971,463 180x50)
        shows SYM_CACHE(m_Input_CACHE := PRG_EVAP.CC13)
    Frame (449,463 180x50)
        shows SYM_CACHE(m_Input_CACHE := PRG_EVAP.CC12)
    Frame (587,564 161x63)
        shows VISU_ALIM_HT_S10(m_Input_HT := PRG_EVAP.SOURCE1)
    Rectangle (606,334 80x40), "M11 :"
    Rectangle (700,334 250x40), "%1.2e mbar", text variable: Global_Variables.PRG_POMPAGE.M11.STATE_Pression
    Polyline (1095,328)
    Polyline (1095,328) (1229,663)
    Polyline (1095,328)
    Polyline (1095,328)
    Frame (1243,607 280x100)
        shows VISU_LIGNE_GAZ_VGAUCHE(m_Input_MACHINE := MACHINE, m_Input_MASSFLOW := PRG_GAZ.DG[2], m_Input_LIGNE_GAZ := PRG_GAZ.LIGNE_GAZ[2])
    Frame (1243,506 280x100)
        shows VISU_LIGNE_GAZ_VGAUCHE(m_Input_MACHINE := MACHINE, m_Input_MASSFLOW := PRG_GAZ.DG[1], m_Input_LIGNE_GAZ := PRG_GAZ.LIGNE_GAZ[1])
    Frame (1239,746 216x103), invisible if: NOT MACHINE.STATE_Manu
        shows VISU_ECOMODE_EVAP()
    Label (390,237 330x63), "Chambre Ouverte", invisible if: PRG_POMPAGE.IN_FE11T
    Image (940,0 400x100), image: MesImages.logo_2012
    Frame (53,647 238x102)
        shows VISU_SWEEP_CHEETAH(m_Input_BALAYAGE := PRG_EVAP.SWEEP1)
    Frame (53,753 260x103)
        shows VISU_CREUSET(m_Input_CREUSET := PRG_EVAP.CRUCIBLE1, m_Input_NUM_CRUCIBLE := 1)
END_VISUALIZATION

// ---- Visualizations/Synoptique/SYN_SERVITUDES.TcVIS
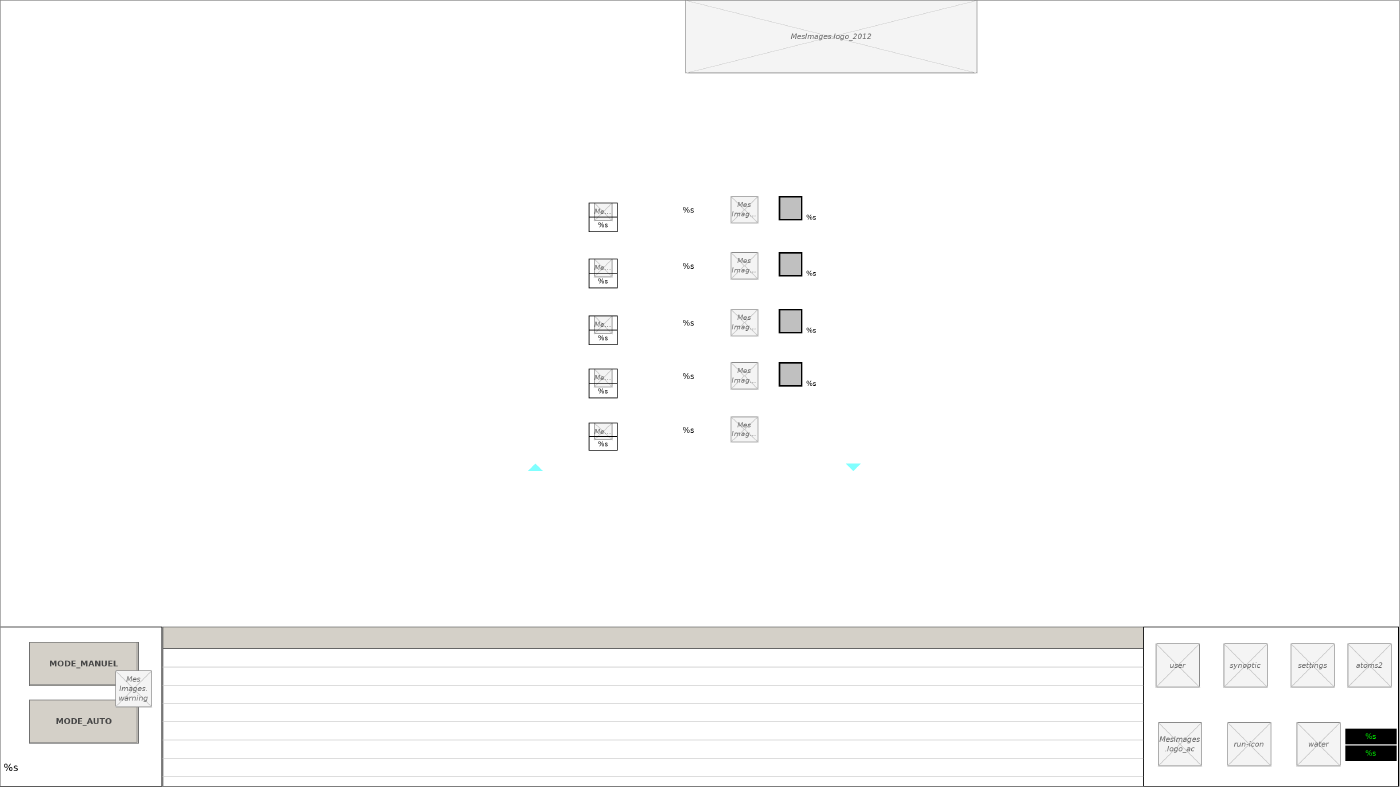
VISUALIZATION SYN_SERVITUDES  // 1920x1080, background image fond_blanc_1280_1024
    Frame (223,860 710x161)
        shows VISU_EV_EXTRAIT()
    Frame (1568,860 352x162)
        shows VISU_BANDEAU(m_Input_MACHINE := Global_Variables.MACHINE)
    Frame (0,860 221x162)
        shows VISU_MODE_MARCHE(m_Input_MACHINE := .MACHINE)
    Polyline (403,450)
    Polyline (403,450)
    Polygon (734,636) (724,646) (744,646)
    Polygon (1170,646) (1160,636) (1180,636)
    Image (940,0 400x100), image: MesImages.logo_2012
    Frame (734,496 438x50)
        shows VISU_LIGNE_EAU(m_Input_LIGNE_EAU := PRG_SERVITUDES.LIGNE_REF[4])
    Frame (734,571 438x47)
        shows VISU_LIGNE_EAU_NO_DEXT(m_Input_LIGNE_EAU := PRG_SERVITUDES.LIGNE_REF[5])
    Frame (734,268 438x50)
        shows VISU_LIGNE_EAU(m_Input_LIGNE_EAU := PRG_SERVITUDES.LIGNE_REF[1])
    Frame (734,345 438x50)
        shows VISU_LIGNE_EAU(m_Input_LIGNE_EAU := PRG_SERVITUDES.LIGNE_REF[2])
    Frame (734,423 438x50)
        shows VISU_LIGNE_EAU(m_Input_LIGNE_EAU := PRG_SERVITUDES.LIGNE_REF[3])
END_VISUALIZATION

// ---- Visualizations/Users/UTIL_CONFIRM.TcVIS
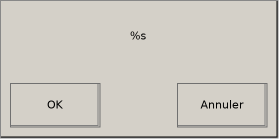
VISUALIZATION UTIL_CONFIRM  // 279x139
VAR_INPUT
	Num_Text:		INT;
END_VAR
VAR_IN_OUT
	OrdreDD:		BOOL;
	Visu:			BOOL;	
END_VAR
    RoundedRectangle (0,0 277x137)
    Textfield (19,6 238x60), "%s", text list: 'TextList_Users_Menu', text index: Num_Text
    Button (10,83 90x44), "OK"
        OnMouseClick: execute { OrdreDD:=(TRUE); }
        OnMouseClick: execute { Visu:=(FALSE); }
    Button (177,83 90x44), "Annuler"
        OnMouseClick: execute { Visu:=(FALSE); }
END_VISUALIZATION

// ---- Visualizations/Users/UTIL_DEFAUT.TcVIS
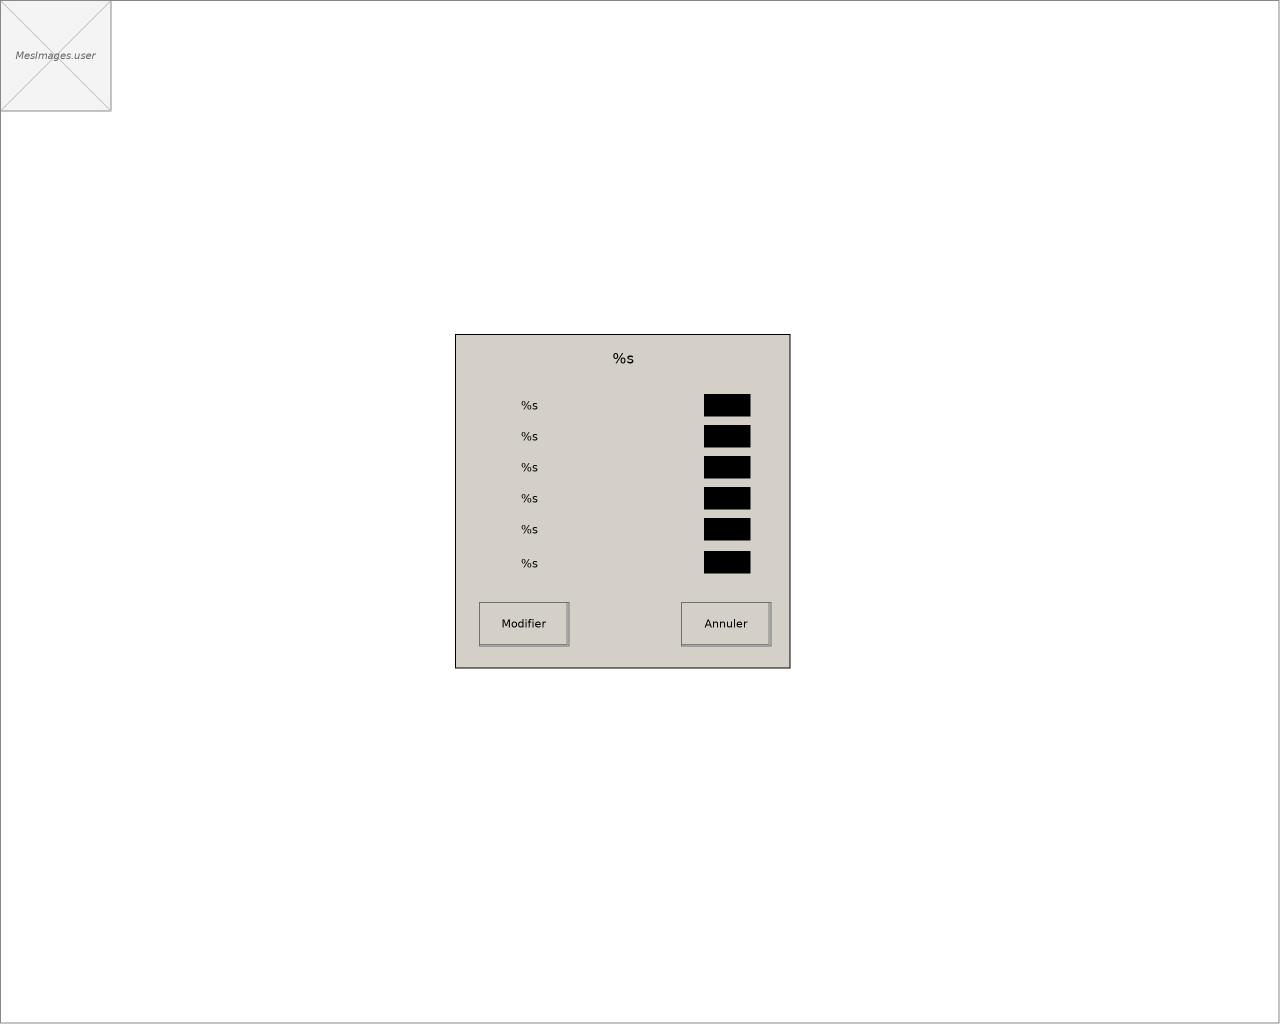
VISUALIZATION UTIL_DEFAUT  // 1280x1024
    Image (0,0 111x111), image: MesImages.user
    RoundedRectangle (455,334 335x334)
    Rectangle (460,344 327x29), "%s", text list: 'TextList_Util_Defaut', text index: 1
    Rectangle (518,422 112x29), "%s", text list: 'TextList_Util_Group', text index: 4
    Rectangle (518,453 112x29), "%s", text list: 'TextList_Util_Group', text index: 5
    Rectangle (518,391 112x29), "%s", text list: 'TextList_Util_Group', text index: 3
    Rectangle (518,484 112x29), "%s", text list: 'TextList_Util_Group', text index: 6
    Rectangle (518,515 112x29), "%s", text list: 'TextList_Util_Group', text index: 7
    Rectangle (518,549 122x29), "%s", text list: 'TextList_Util_Group', text index: 8
    Rectangle (704,394 46x22), "Oui", colour toggle: Global_Variables.PRG_USER.GROUP_TEMP.PROGRAMMATION
        toggle Global_Variables.PRG_USER.GROUP_TEMP.PROGRAMMATION
    Rectangle (704,425 46x22), "Oui", colour toggle: Global_Variables.PRG_USER.GROUP_TEMP.MAINTENANCE
        toggle Global_Variables.PRG_USER.GROUP_TEMP.MAINTENANCE
    Rectangle (704,456 46x22), "Oui", colour toggle: Global_Variables.PRG_USER.GROUP_TEMP.SUPERVISEUR
        toggle Global_Variables.PRG_USER.GROUP_TEMP.SUPERVISEUR
    Rectangle (704,487 46x22), "Oui", colour toggle: Global_Variables.PRG_USER.GROUP_TEMP.PRODUCTION
        toggle Global_Variables.PRG_USER.GROUP_TEMP.PRODUCTION
    Rectangle (704,518 46x22), "Oui", colour toggle: Global_Variables.PRG_USER.GROUP_TEMP.CONF_MACHINE
        toggle Global_Variables.PRG_USER.GROUP_TEMP.CONF_MACHINE
    Rectangle (704,551 46x22), "Oui", colour toggle: Global_Variables.PRG_USER.GROUP_TEMP.FONCTION_SA
        toggle Global_Variables.PRG_USER.GROUP_TEMP.FONCTION_SA
    Button (479,602 90x44), "Modifier"
        toggle PRG_USER.DD_mod_def2
        OnMouseClick: change screen: UTIL_MENU
    Button (681,602 90x44), "Annuler"
        OnMouseClick: change screen: UTIL_MENU
END_VISUALIZATION

// ---- Visualizations/Users/UTIL_DELOG.TcVIS
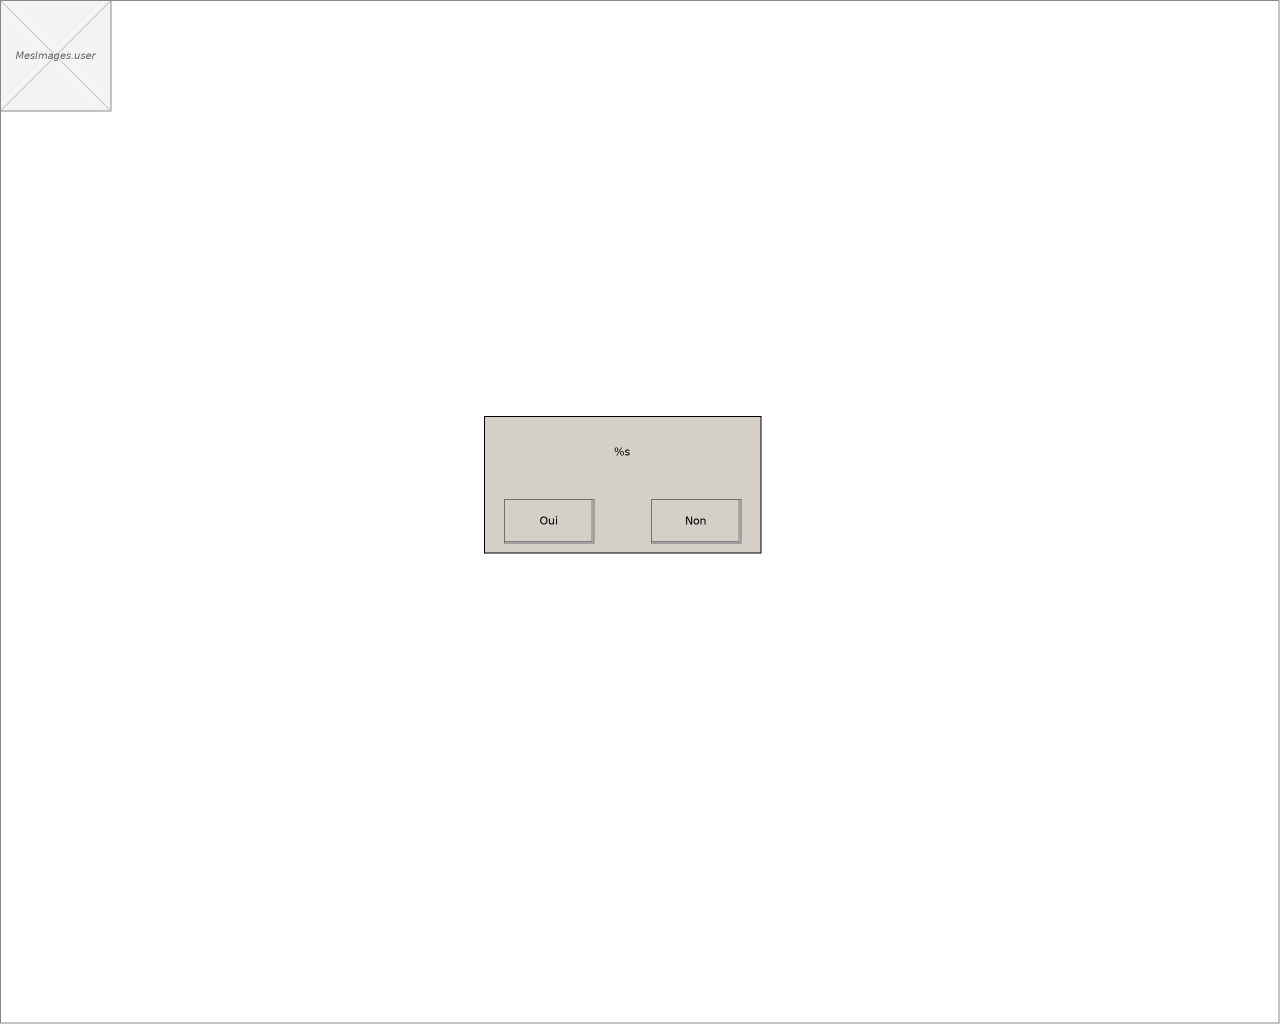
VISUALIZATION UTIL_DELOG  // 1280x1024
    Image (0,0 111x111), image: MesImages.user
    RoundedRectangle (484,416 277x137)
    Textfield (503,422 238x60), "%s", text list: 'TextList_Users_Menu', text index: 3
    Button (504,499 90x44), "Oui"
        toggle PRG_USER.DD_DELOG
        OnMouseClick: change screen: UTIL_MENU
    Button (651,499 90x44), "Non"
        OnMouseClick: change screen: UTIL_MENU
END_VISUALIZATION

// ---- Visualizations/Users/UTIL_GROUP.TcVIS
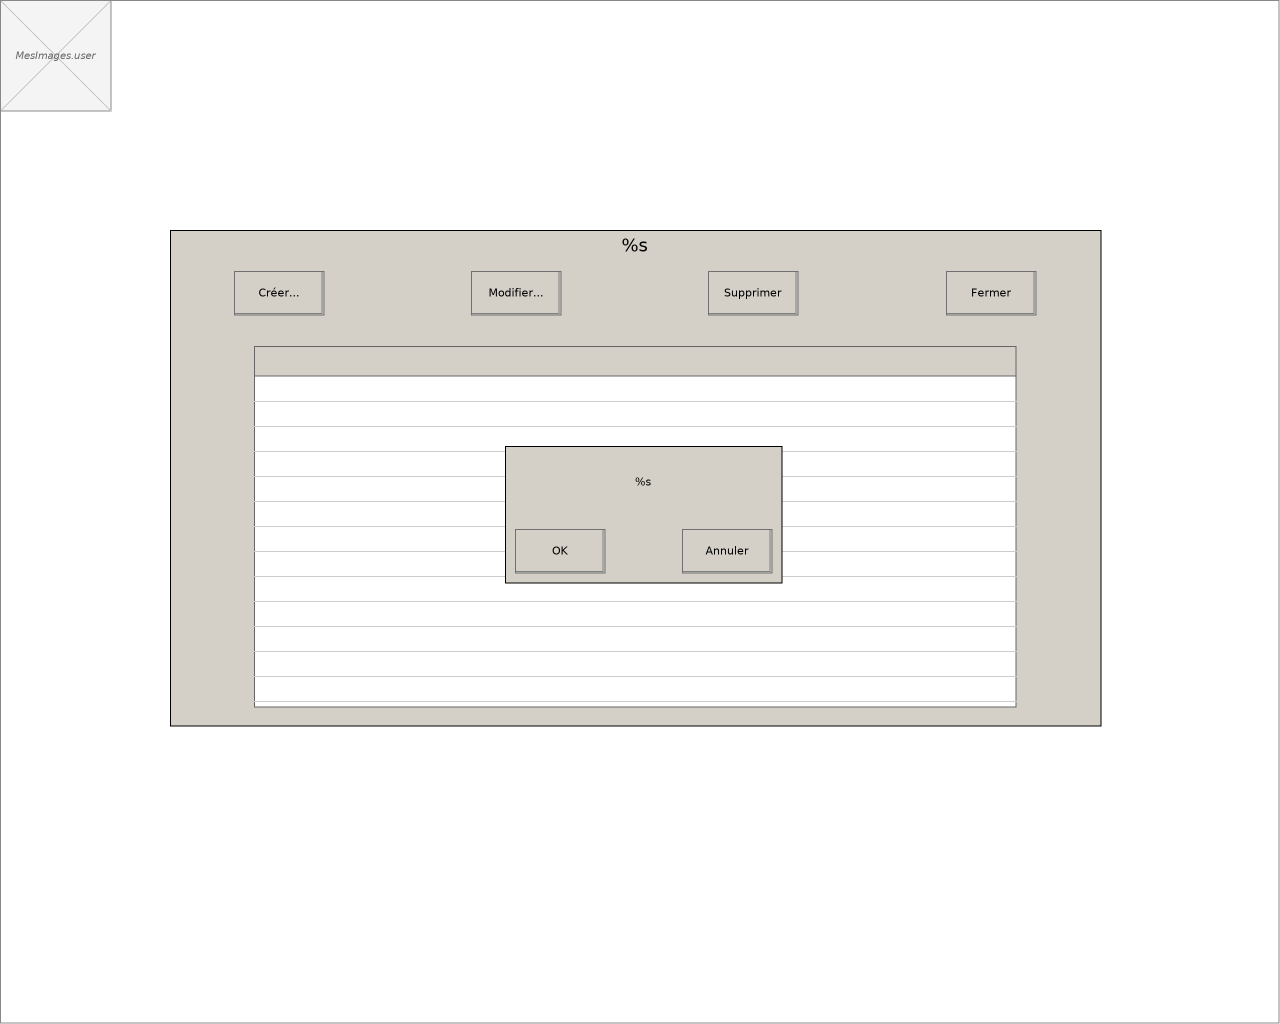
VISUALIZATION UTIL_GROUP  // 1280x1024
    RoundedRectangle (170,230 931x496)
    Image (0,0 111x111), image: MesImages.user
    Table (254,346 762x361), data array: PRG_USER.TBL_GROUP
        p1137915858: PRG_USER.LIGNE_GROUP
        p3854506369: PRG_USER.TBL_GROUP[INDEX].NOM
        p1892666644: PRG_USER.TBL_GROUP[INDEX].PROGRAMMATION
        p338671338: PRG_USER.TBL_GROUP[INDEX].MAINTENANCE
        p2170511999: PRG_USER.TBL_GROUP[INDEX].SUPERVISEUR
        p3723444502: PRG_USER.TBL_GROUP[INDEX].PRODUCTION
        p1218418051: PRG_USER.TBL_GROUP[INDEX].CONF_MACHINE
        p746581629: PRG_USER.TBL_GROUP[INDEX].FONCTION_SA
        p3104783080: PRG_USER.TBL_GROUP[INDEX].CONF_TRF
        p2501879983: PRG_USER.TBL_GROUP[INDEX].MODIF_ENLIGNE
        p7306298: PRG_USER.TBL_GROUP[INDEX].ARCHIVE_EV
        p1933151965: PRG_USER.TBL_GROUP[INDEX].DECONSIGNATION
        p2232123230: Nom du groupe
        p511219082: Pro. Ed
        p1755163831: Maint.
        p4092479075: Superv.
        p2237128397: Prod.
        p505689113: Conf.
        p1757482276: FoncSA.
    Textfield (231,233 808x25), "%s", text list: 'TextList_Util_Userlist', text index: 5
    Button (234,271 90x44), "Créer...", invisible if: PRG_USER.STOP_GROUP
        toggle PRG_USER.DD_EFFACE_NEW2
        OnMouseClick: change screen: UTIL_NEW_GROUP
    Button (471,271 90x44), "Modifier...", input disabled if: NOT PRG_USER.AUT_MOD_GRP
        toggle PRG_USER.DD_mod_group1
        OnMouseClick: change screen: UTIL_MOD_GROUP
    Button (708,271 90x44), "Supprimer", input disabled if: NOT PRG_USER.AUT_MOD_GRP
        toggle PRG_USER.VISU_FEN4
    Button (946,271 90x44), "Fermer", input disabled if: PRG_USER.VISU_FEN4
        OnMouseClick: change screen: UTIL_MENU
    Frame (505,446 280x139), invisible if: NOT PRG_USER.VISU_FEN4
        shows UTIL_CONFIRM(Num_Text := 19, OrdreDD := PRG_USER.DD_DEL_GROUP, Visu := PRG_USER.VISU_FEN4)
END_VISUALIZATION

// ---- Visualizations/Users/UTIL_LOG.TcVIS
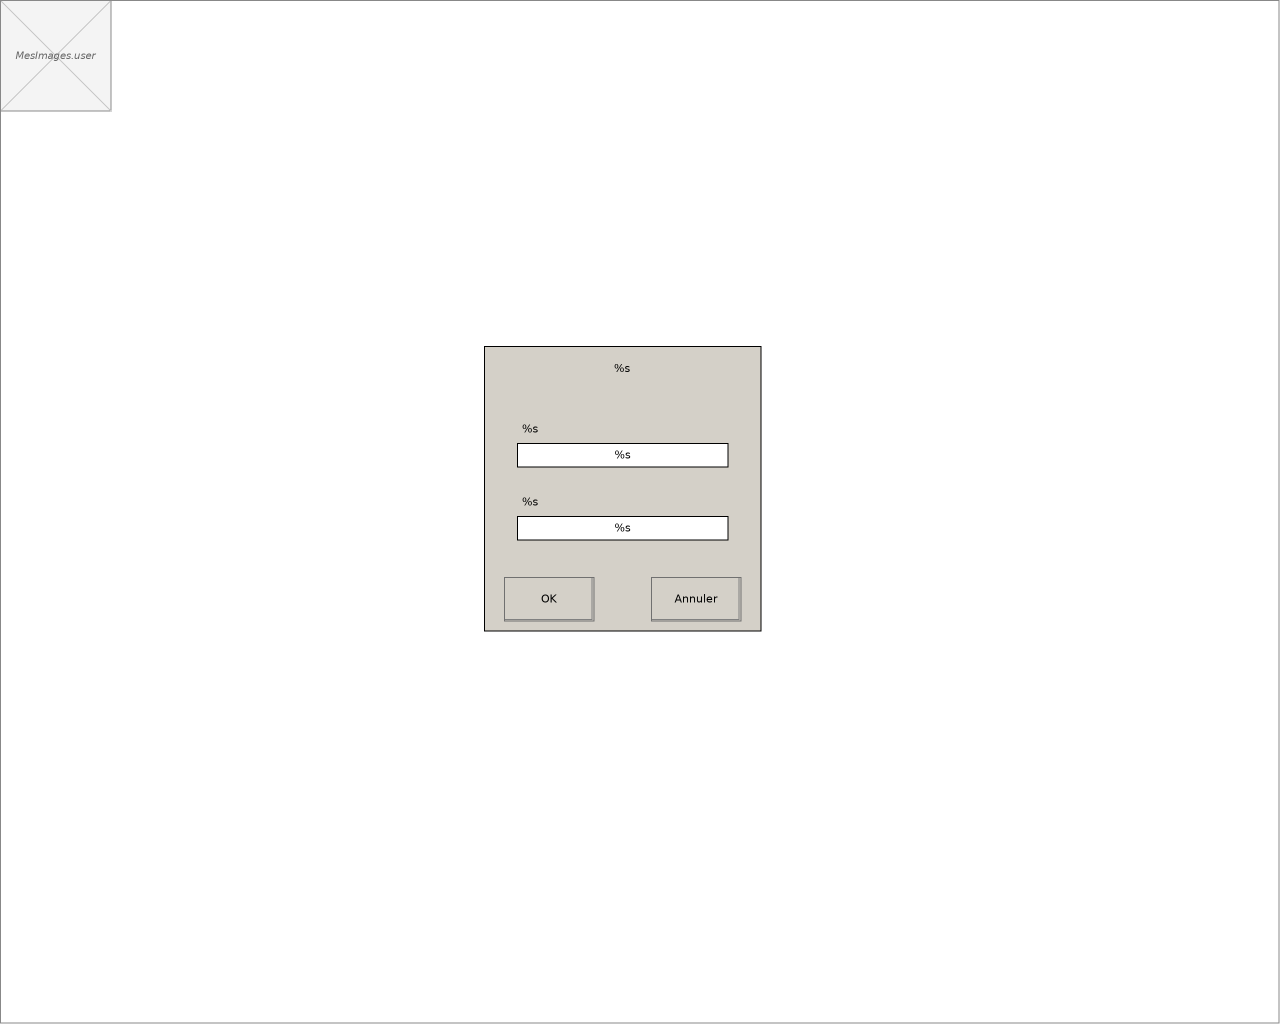
VISUALIZATION UTIL_LOG  // 1280x1024
    Image (0,0 111x111), image: MesImages.user
    RoundedRectangle (484,346 277x285)
    Textfield (503,356 238x25), "%s", text list: 'TextList_Users_Menu', text index: 4
    Button (504,577 90x44), "OK"
        toggle PRG_USER.DD_LOG
        OnMouseClick: change screen: UTIL_MENU
    Button (651,577 90x44), "Annuler"
        OnMouseClick: change screen: UTIL_MENU
    Rectangle (517,443 211x24), "%s", text variable: PRG_USER.LOG_TEMP
        OnMouseClick: write the text variable via InputWithLimits
    Rectangle (517,516 211x24), "%s", text variable: PRG_USER.PASS_TEMP_DISPLAY
        OnMouseClick: write PRG_USER.PASS_TEMP via InputWithLimits, password
    Textfield (519,419 126x20), "%s", text list: 'TextList_Users_Menu', text index: 5
    Textfield (519,492 126x20), "%s", text list: 'TextList_Users_Menu', text index: 6
END_VISUALIZATION

// ---- Visualizations/Users/UTIL_MENU.TcVIS
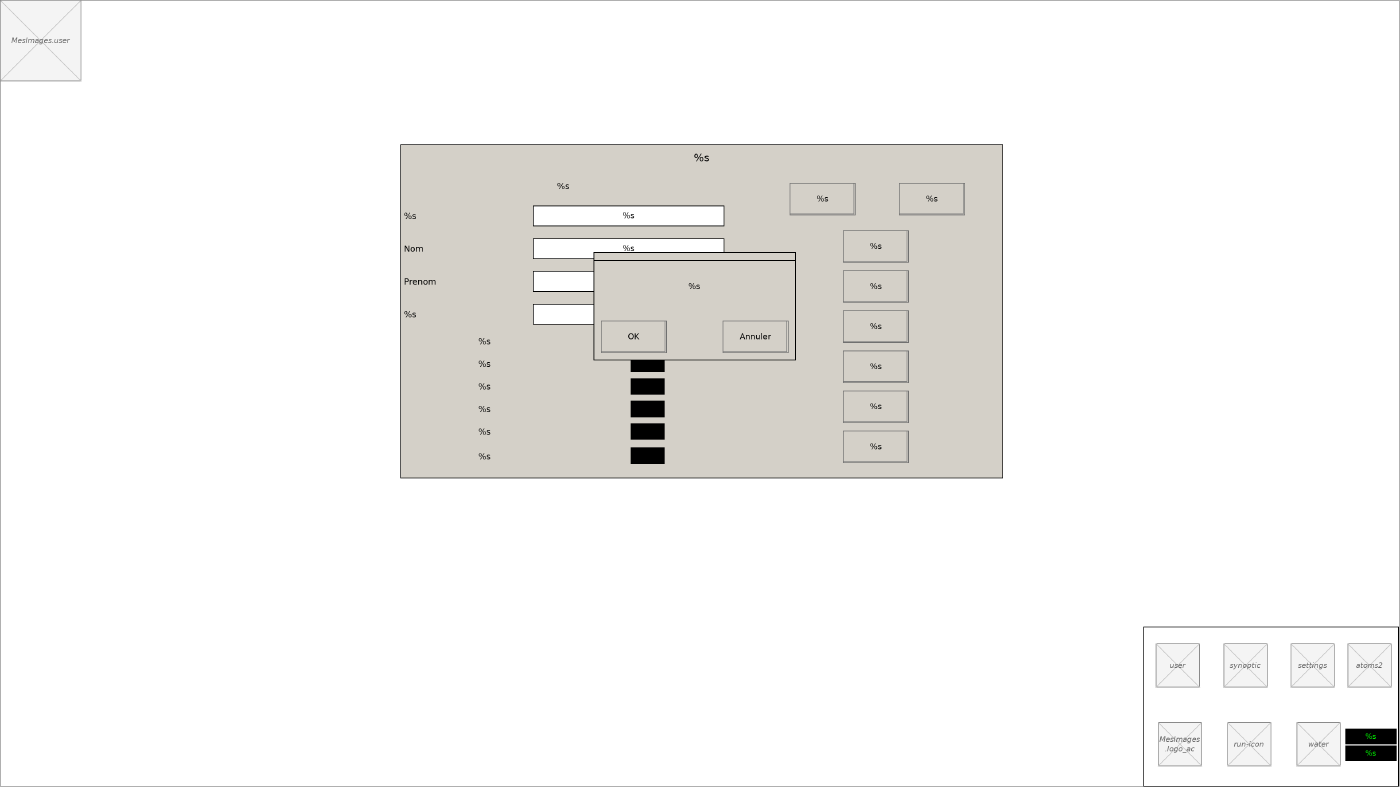
VISUALIZATION UTIL_MENU  // 1920x1080
    Image (0,0 111x111), image: MesImages.user
    RoundedRectangle (549,198 826x458)
    Rectangle (553,202 819x29), "%s", text list: 'TextList_Users_Menu', text index: 1
    Rectangle (731,282 262x28), "%s", text variable: PRG_USER.ACTU_USER.LOGIN
    Rectangle (552,241 441x29), "%s", text list: 'TextList_Users_Menu', text index: 7
    Rectangle (551,282 173x29), "%s", text list: 'TextList_Users_Menu', text index: 5
    Rectangle (551,327 173x29), "Nom"
    Rectangle (551,372 173x29), "Prenom"
    Rectangle (731,327 262x28), "%s", text variable: PRG_USER.ACTU_USER.NOM
    Rectangle (731,372 262x28), "%s", text variable: PRG_USER.ACTU_USER.PRENOM
    Rectangle (551,417 173x29), "%s", text list: 'TextList_Users_Menu', text index: 8
    Rectangle (731,417 262x28), "%s", text variable: PRG_USER.ACTU_USER.GROUPE
        OnMouseClick: write the text variable via VisuDialogs.Keypad
    Rectangle (653,485 112x29), "%s", text list: 'TextList_Util_Group', text index: 4
    Rectangle (653,516 112x29), "%s", text list: 'TextList_Util_Group', text index: 5
    Rectangle (653,454 112x29), "%s", text list: 'TextList_Util_Group', text index: 3
    Rectangle (653,547 112x29), "%s", text list: 'TextList_Util_Group', text index: 6
    Rectangle (653,578 112x29), "%s", text list: 'TextList_Util_Group', text index: 7
    Rectangle (653,612 122x29), "%s", text list: 'TextList_Util_Group', text index: 8
    Rectangle (865,457 46x22), "Oui", colour toggle: PRG_USER.ACTU_USER.PROGRAMMATION
    Rectangle (865,488 46x22), "Oui", colour toggle: PRG_USER.ACTU_USER.MAINTENANCE
    Rectangle (865,519 46x22), "Oui", colour toggle: PRG_USER.ACTU_USER.SUPERVISEUR
    Rectangle (865,550 46x22), "Oui", colour toggle: PRG_USER.ACTU_USER.PRODUCTION
    Rectangle (865,581 46x22), "Oui", colour toggle: PRG_USER.ACTU_USER.CONF_MACHINE
    Rectangle (865,614 46x22), "Oui", colour toggle: PRG_USER.ACTU_USER.FONCTION_SA
    Button (1083,251 90x44), "%s", input disabled if: PRG_USER.UTIL_EC, text list: 'TextList_Users_Menu', text index: 9
        toggle PRG_USER.DD_LOG1
        OnMouseClick: change screen: UTIL_LOG
    Button (1233,251 90x44), "%s", input disabled if: MAIN.VAR_INVISIBLE_DELOG, text list: 'TextList_Users_Menu', text index: 10
        OnMouseClick: change screen: UTIL_DELOG
    Button (1156,316 90x44), "%s", input disabled if: NOT PRG_USER.ACTU_USER.SUPERVISEUR, text list: 'TextList_Users_Menu', text index: 11
        toggle PRG_USER.DD_mod_def1
        OnMouseClick: change screen: UTIL_DEFAUT
    Button (1156,371 90x44), "%s", input disabled if: NOT PRG_USER.ACTU_USER.SUPERVISEUR, text list: 'TextList_Users_Menu', text index: 12
        OnMouseClick: change screen: UTIL_USER
    Button (1156,426 90x44), "%s", input disabled if: NOT PRG_USER.ACTU_USER.SUPERVISEUR, text list: 'TextList_Users_Menu', text index: 13
        OnMouseClick: change screen: UTIL_GROUP
    Button (1156,481 90x44), "%s", input disabled if: PRG_USER.LOAD_EC OR NOT PRG_USER.ACTU_USER.SUPERVISEUR OR PRG_USER.SAVE_EC, text list: 'TextList_Users_Menu', text index: 14
        toggle PRG_USER.VISU_FEN1
    Button (1156,536 90x44), "%s", input disabled if: PRG_User.SAVE_EC OR NOT PRG_User.ACTU_USER.SUPERVISEUR OR PRG_User.LOAD_EC, text list: 'TextList_Users_Menu', text index: 15
        toggle PRG_USER.VISU_FEN2
    Button (1156,591 90x44), "%s", input disabled if: NOT PRG_USER.ACTU_USER.SUPERVISEUR, text list: 'TextList_Users_Menu', text index: 16
        toggle PRG_USER.DD_mod_def1
        OnMouseClick: change screen: UTIL_OPT
    Frame (814,346 278x137), invisible if: NOT PRG_USER.VISU_FEN1
        shows UTIL_CONFIRM(Num_Text := 20, OrdreDD := PRG_USER.DD_load, Visu := PRG_USER.VISU_FEN1)
    Frame (814,357 278x137), invisible if: NOT PRG_USER.VISU_FEN2
        shows UTIL_CONFIRM(Num_Text := 17, OrdreDD := PRG_USER.DD_sauv, Visu := PRG_USER.VISU_FEN2)
    Frame (1568,860 352x162)
        shows VISU_BANDEAU(m_Input_MACHINE := Global_Variables.MACHINE)
END_VISUALIZATION

// ---- Visualizations/Users/UTIL_MOD_GROUP.TcVIS
